# EPICS StreamDevice protocol: protocols/ai_waterfall.proto
Terminator = LF;
ExtraInput = Ignore;
ReplyTimeout = 5000;

setAiWaterfall {
        out "ai_waterfall %d";
        in;
}
